// SIMATIC S7-200 project (STEP 7-Micro/WIN), CPU 224XP REL 02.01

ORGANIZATION_BLOCK 主程序:OB1
TITLE=程序注释
BEGIN
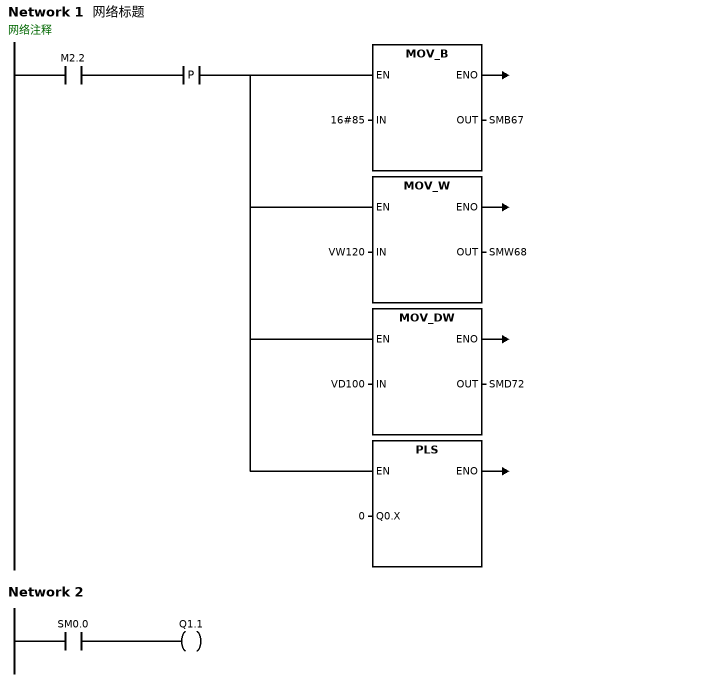
Network 1 // 网络标题
// 网络注释
LD     M2.2
EU
MOVB   16#85, SMB67
MOVW   VW120, SMW68
MOVD   VD100, SMD72
PLS    0
Network 2
LD     SM0.0
=      Q1.1
END_ORGANIZATION_BLOCK
